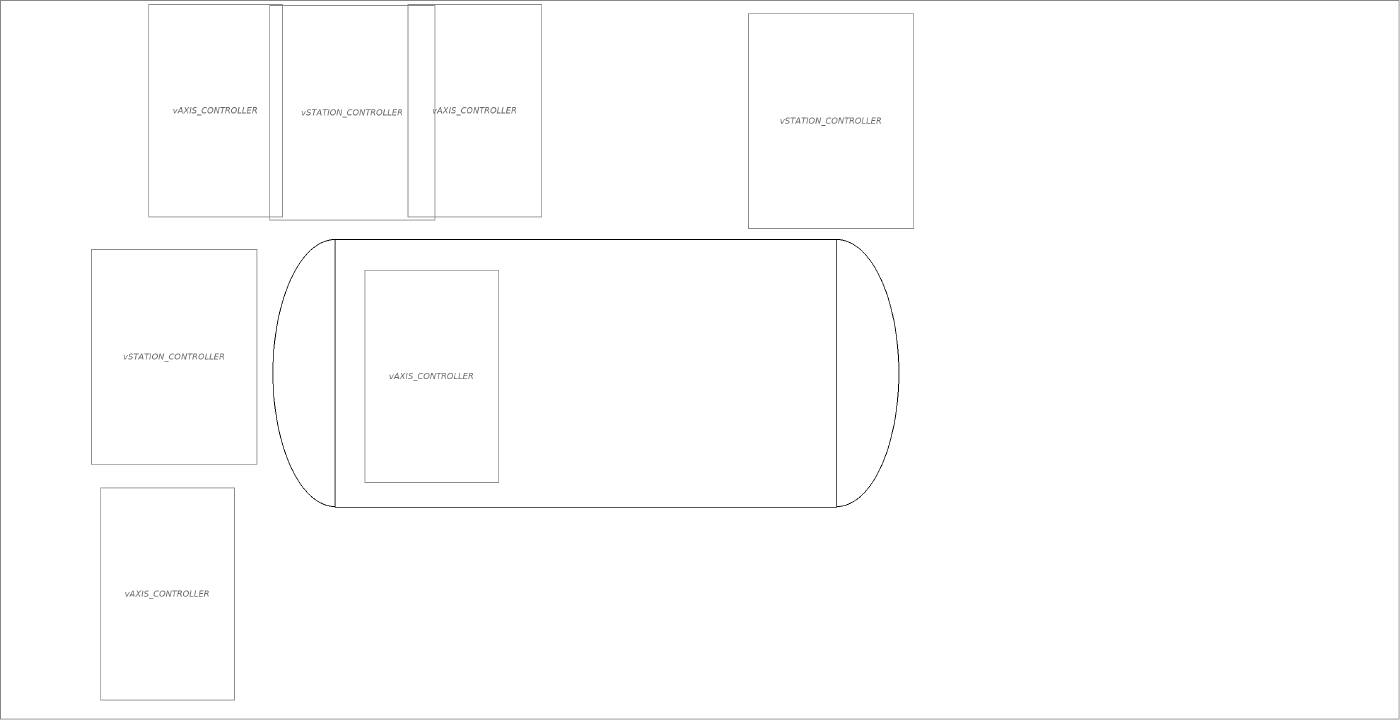
VISUALIZATION vMACHINE  // 1690x870
    Frame (110,301 200x260)
        shows vSTATION_CONTROLLER(vSTATION := fbFEEDER)
    Frame (325,6 200x260)
        shows vSTATION_CONTROLLER(vSTATION := fbSEPARATE1)
    Frame (903,16 200x260)
        shows vSTATION_CONTROLLER(vSTATION := fbSEPARATE2)
    Ellipse (329,289 150x323)
    Ellipse (935,289 150x323)
    Rectangle (404,289 606x324)
    Frame (440,326 162x257)
        shows vAXIS_CONTROLLER(vAXIS := MAIN_CONV)
    Frame (121,589 162x257)
        shows vAXIS_CONTROLLER(vAXIS := SUP_CONV)
    Frame (492,5 162x257)
        shows vAXIS_CONTROLLER(vAXIS := PRESS1B)
    Frame (179,5 162x257)
        shows vAXIS_CONTROLLER(vAXIS := PRESS1A)
END_VISUALIZATION

(* stored: Version 1.1.0.1, ProductVersion 3.1.4024.12
   Visu vMACHINE: Id {3deaac7f-3d0e-48ef-a7db-42e8b819f786} *)
